/// determines whether the actual speed (ABS value) is within the target-speed window
FUNCTION F_SpeedReached : BOOL
VAR_INPUT
	/// actual speed
	fActualSpeed: LREAL;
	/// target speed
	fTargetSpeed: LREAL;
	/// Override for axis and spindle
	fOverride: LREAL;
END_VAR

F_SpeedReached := F_SpeedWindowReached(fToleranceFactor:=0, fActualSpeed:=fActualSpeed, fTargetSpeed:=fTargetSpeed, fOverride:=fOverride);

END_FUNCTION

(* stored: Version 1.1.0.1, ProductVersion 3.1.4020.12
   POU F_SpeedReached: Id {e8f3e6cf-3707-4a0f-9892-9a3076f2927a}, SpecialFunc None *)
